(* IEC 61131-3 sources: cc_kush_rewrite/POUs/Conveyor/FC, 4 files *)

(* ---- FC_Conveyor_EmergencyStop.st ---- *)
FUNCTION FC_Conveyor_EmergencyStop : BOOL
VAR_INPUT
	Conveyor : REFERENCE TO ST_ConveyorPrefabricated;
END_VAR
VAR
	j : INT;
END_VAR

// Аварийная остановка всех моторов конвейера
FOR j := 1 TO 2 DO
	Conveyor.MotorConveyor[j].qxKM_Power := FALSE;
	Conveyor.MotorConveyor[j].VFD.qxStart := FALSE;
	Conveyor.MotorConveyor[j].VFD.Frequency.rTargetFrequency := 0.0;
	Conveyor.MotorConveyor[j].VFD.qrOutFrequency := 0.0;
END_FOR

// Активация тормоза
Conveyor.qxBreakerConveyor := FALSE;

FC_Conveyor_EmergencyStop := TRUE;

END_FUNCTION

(* ---- FC_Conveyor_GetErrorCommon.st ---- *)
FUNCTION FC_Conveyor_GetErrorCommon : BOOL
VAR_INPUT
	Conveyor : REFERENCE TO ST_ConveyorPrefabricated;
END_VAR
VAR
END_VAR
FC_Conveyor_GetErrorCommon :=
	FC_Conveyor_GetErrorSensors(Conveyor := Conveyor)
	OR FC_Conveyor_GetErrorMotor(motor := Conveyor.MotorConveyor[1])
	OR FC_Conveyor_GetErrorMotor(motor := Conveyor.MotorConveyor[2]);

END_FUNCTION

(* ---- FC_Conveyor_GetErrorMotor.st ---- *)
FUNCTION FC_Conveyor_GetErrorMotor : BOOL
VAR_INPUT
	motor : REFERENCE TO ST_MotorWithFeedback;
END_VAR
VAR
END_VAR
FC_Conveyor_GetErrorMotor := (
	motor.VFD.fbStateFailure.qxInvertedSignal // Ошибка ЧРП (NC: TRUE=норма, инвертированный=TRUE=ошибка)
	OR motor.VFD.xStateFailureLocal // Ошибка ЧРП, полученная программным путем
	OR motor.VFD.fbRangeDiagnostic.qxCriticalActive // Критическое значение тока эл. двигателя
	OR NOT motor.fbStatorOverheat.qxSignal // Перегрев статора (1 - норма, 0 - перегрев)
);

END_FUNCTION

(* ---- FC_Conveyor_GetErrorSensors.st ---- *)
FUNCTION FC_Conveyor_GetErrorSensors : BOOL
VAR_INPUT
	Conveyor : REFERENCE TO ST_ConveyorPrefabricated;
END_VAR
VAR
END_VAR
FC_Conveyor_GetErrorSensors := (
	// Контроль схода ленты - тревога
	FC_Sensor_CheckZQAlarm(fbZQAlarm := Conveyor.fbZQAlarm)
	// Кабель-тросовый выключатель
	OR FC_Sensor_CheckHQ(fbHQ_IsOk := Conveyor.fbHQ_IsOk)
	// Контроль ограждения барабана
	OR FC_Sensor_CheckSQ(fbSQ_IsOk := Conveyor.fbSQ_IsOk)
	// Контроль заштыбовки
	OR FC_Sensor_CheckGS(fbGS := Conveyor.fbGS1)
	// Контроль продольного разрыва ленты
	OR FC_Sensor_CheckYS(fbYS := Conveyor.fbYS1)
	// Обнаружение металла
	OR FC_Sensor_CheckYE(fbYE := Conveyor.fbYE1)
);

END_FUNCTION
